PROGRAM MAIN_1
VAR
	execute AT %I* : BOOL;
	trigger : R_TRIG;
	
	newBundle AT %M* : Bundle;
	bundlesQueue : ARRAY[0..CONSTS.maxQueue] OF Bundle;
END_VAR

(*
Area 3 contains <n> buffers, each index contains 6 conveyors
	this allows each buffer to carry up to a theoretical maximum of 6 bundles - realistically this will be limited to 3

implementation:
	each buffer stores 6 iterators (1 for each conveyor) to point to an element in bundlesQueue, and a master conveyor mode request
	compute the master request for the conveyors within a buffer, then use the buffer master request to link all buffers
*)

METHOD PRIVATE blocks : BOOL
VAR_INPUT
END_VAR
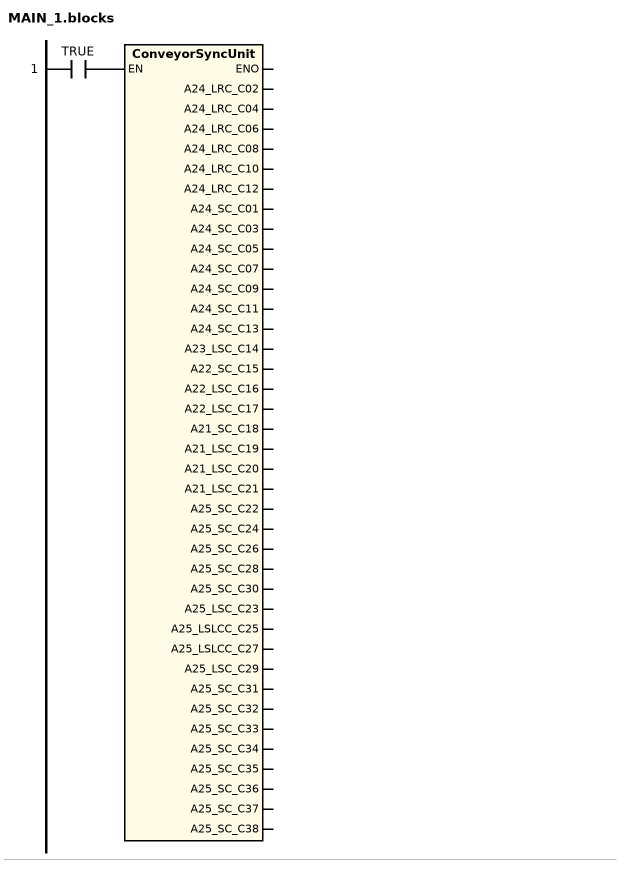
// NETWORK 1
ConveyorSyncUnit();
END_METHOD

METHOD PRIVATE receive : BOOL
VAR_INPUT
END_VAR
VAR
	i : DINT;
END_VAR
FOR i:=0 TO CONSTS.maxQueue BY 1 DO
	
	IF NOT BundleIsValid(bundlesQueue[i]) THEN
		bundlesQueue[i] := newBundle;
		
		receive := TRUE;
		EXIT;
	END_IF
	
END_FOR
END_METHOD

END_PROGRAM

(* stored: Version 1.1.0.1, ProductVersion 3.1.4024.11
   POU MAIN_1: Id {e8fe96bb-13b3-49a8-979b-e8b7929eb562}, SpecialFunc None
   Method blocks: Id {5746b797-156b-48da-9013-04c0b6442aec}
   Method receive: Id {cf11b485-0a7a-43ca-9ace-da02f245f576} *)
